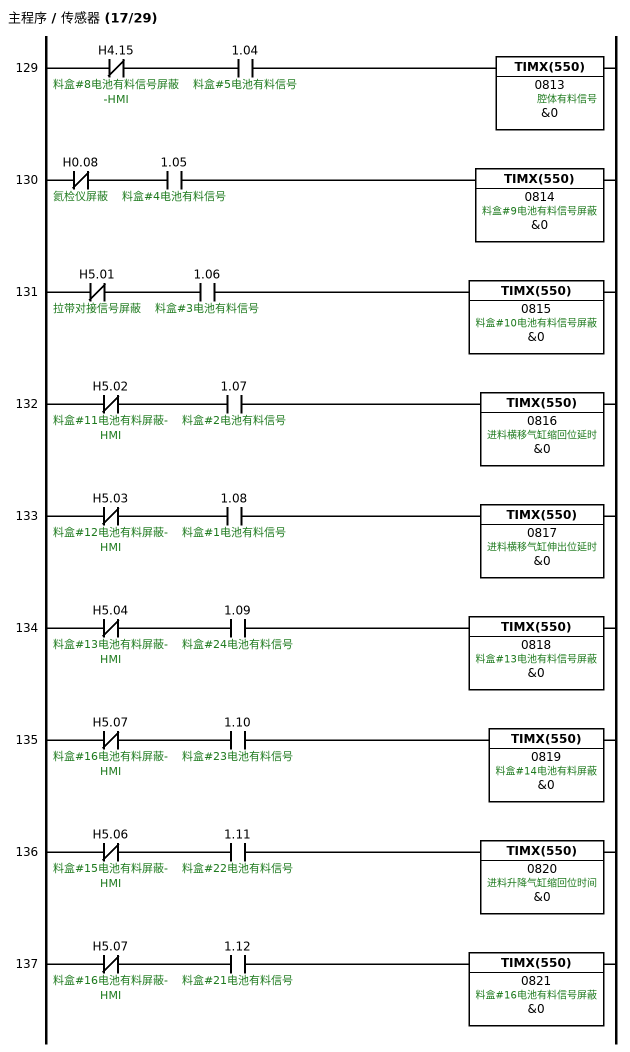
; [picture p24: 主程序 / 传感器, rungs 129-137]
; rung 129
LDNOT H4.15  ; 料盒#8电池有料信号屏蔽-HMI
AND 1.04  ; 料盒#5电池有料信号
TIMX(550) 0813 &0  ; 腔体有料信号
; rung 130
LDNOT H0.08  ; 氦检仪屏蔽
AND 1.05  ; 料盒#4电池有料信号
TIMX(550) 0814 &0  ; 料盒#9电池有料信号屏蔽
; rung 131
LDNOT H5.01  ; 拉带对接信号屏蔽
AND 1.06  ; 料盒#3电池有料信号
TIMX(550) 0815 &0  ; 料盒#10电池有料信号屏蔽
; rung 132
LDNOT H5.02  ; 料盒#11电池有料屏蔽-HMI
AND 1.07  ; 料盒#2电池有料信号
TIMX(550) 0816 &0  ; 进料横移气缸缩回位延时
; rung 133
LDNOT H5.03  ; 料盒#12电池有料屏蔽-HMI
AND 1.08  ; 料盒#1电池有料信号
TIMX(550) 0817 &0  ; 进料横移气缸伸出位延时
; rung 134
LDNOT H5.04  ; 料盒#13电池有料屏蔽-HMI
AND 1.09  ; 料盒#24电池有料信号
TIMX(550) 0818 &0  ; 料盒#13电池有料信号屏蔽
; rung 135
LDNOT H5.07  ; 料盒#16电池有料屏蔽-HMI
AND 1.10  ; 料盒#23电池有料信号
TIMX(550) 0819 &0  ; 料盒#14电池有料屏蔽
; rung 136
LDNOT H5.06  ; 料盒#15电池有料屏蔽-HMI
AND 1.11  ; 料盒#22电池有料信号
TIMX(550) 0820 &0  ; 进料升降气缸缩回位时间
; rung 137
LDNOT H5.07  ; 料盒#16电池有料屏蔽-HMI
AND 1.12  ; 料盒#21电池有料信号
TIMX(550) 0821 &0  ; 料盒#16电池有料信号屏蔽

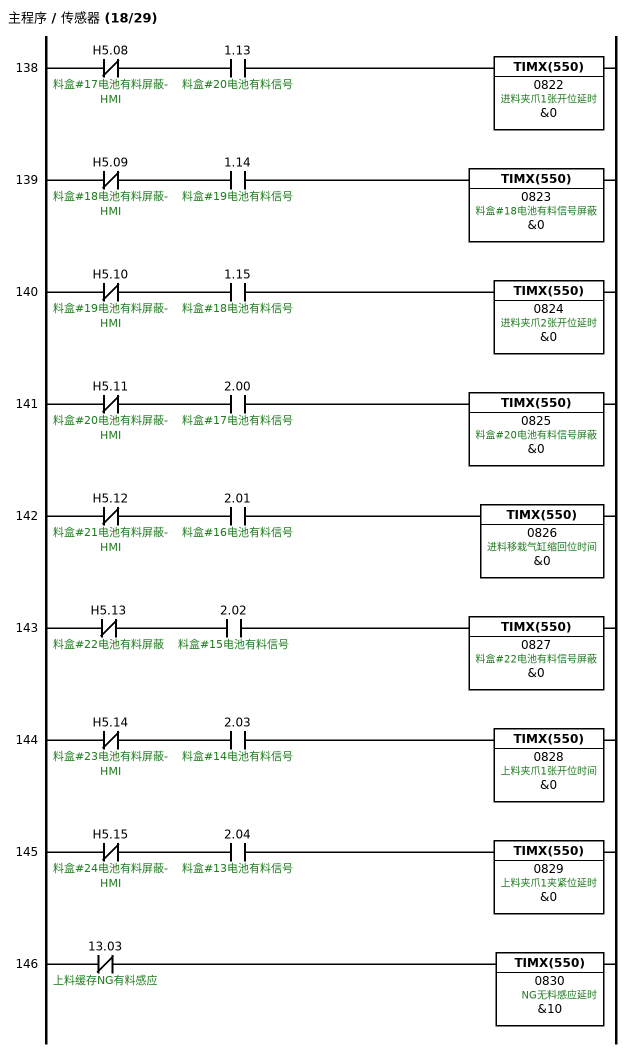
; rung 138
LDNOT H5.08  ; 料盒#17电池有料屏蔽-HMI
AND 1.13  ; 料盒#20电池有料信号
TIMX(550) 0822 &0  ; 进料夹爪1张开位延时
; rung 139
LDNOT H5.09  ; 料盒#18电池有料屏蔽-HMI
AND 1.14  ; 料盒#19电池有料信号
TIMX(550) 0823 &0  ; 料盒#18电池有料信号屏蔽
; rung 140
LDNOT H5.10  ; 料盒#19电池有料屏蔽-HMI
AND 1.15  ; 料盒#18电池有料信号
TIMX(550) 0824 &0  ; 进料夹爪2张开位延时
; rung 141
LDNOT H5.11  ; 料盒#20电池有料屏蔽-HMI
AND 2.00  ; 料盒#17电池有料信号
TIMX(550) 0825 &0  ; 料盒#20电池有料信号屏蔽
; rung 142
LDNOT H5.12  ; 料盒#21电池有料屏蔽-HMI
AND 2.01  ; 料盒#16电池有料信号
TIMX(550) 0826 &0  ; 进料移栽气缸缩回位时间
; rung 143
LDNOT H5.13  ; 料盒#22电池有料屏蔽
AND 2.02  ; 料盒#15电池有料信号
TIMX(550) 0827 &0  ; 料盒#22电池有料信号屏蔽
; rung 144
LDNOT H5.14  ; 料盒#23电池有料屏蔽-HMI
AND 2.03  ; 料盒#14电池有料信号
TIMX(550) 0828 &0  ; 上料夹爪1张开位时间
; rung 145
LDNOT H5.15  ; 料盒#24电池有料屏蔽-HMI
AND 2.04  ; 料盒#13电池有料信号
TIMX(550) 0829 &0  ; 上料夹爪1夹紧位延时
; rung 146
LDNOT 13.03  ; 上料缓存NG有料感应
TIMX(550) 0830 &10  ; NG无料感应延时

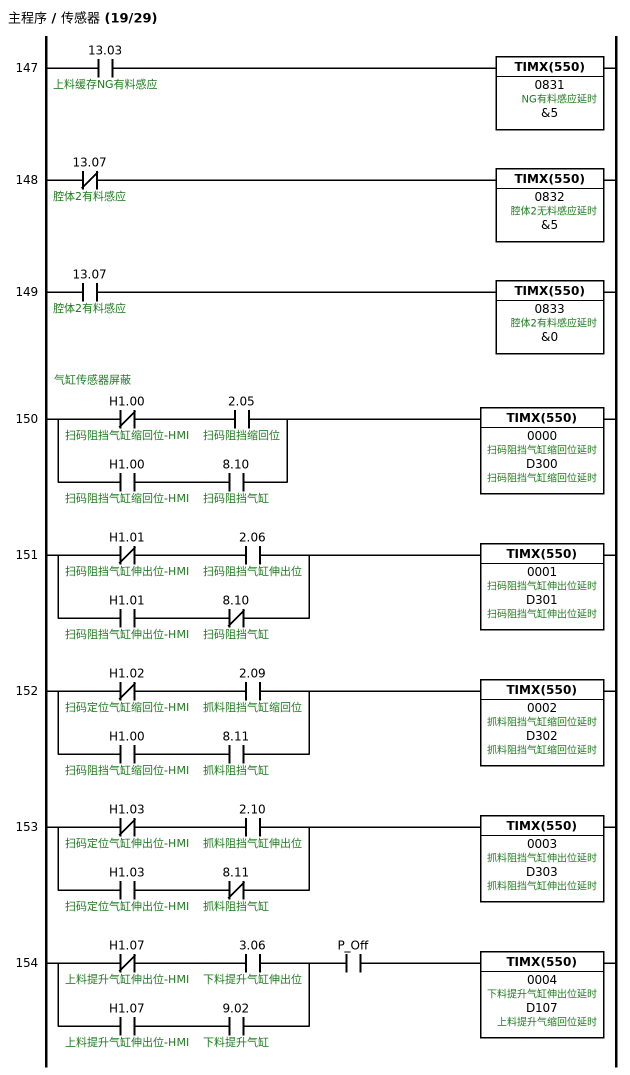
; rung 147
LD 13.03  ; 上料缓存NG有料感应
TIMX(550) 0831 &5  ; NG有料感应延时
; rung 148
LDNOT 13.07  ; 腔体2有料感应
TIMX(550) 0832 &5  ; 腔体2无料感应延时
; rung 149
LD 13.07  ; 腔体2有料感应
TIMX(550) 0833 &0  ; 腔体2有料感应延时
; rung 150: 气缸传感器屏蔽
LDNOT H1.00  ; 扫码阻挡气缸缩回位-HMI
AND 2.05  ; 扫码阻挡缩回位
LD H1.00  ; 扫码阻挡气缸缩回位-HMI
AND 8.10  ; 扫码阻挡气缸
ORLD
TIMX(550) 0000 D300  ; 扫码阻挡气缸缩回位延时
; rung 151
LDNOT H1.01  ; 扫码阻挡气缸伸出位-HMI
AND 2.06  ; 扫码阻挡气缸伸出位
LD H1.01  ; 扫码阻挡气缸伸出位-HMI
ANDNOT 8.10  ; 扫码阻挡气缸
ORLD
TIMX(550) 0001 D301  ; 扫码阻挡气缸伸出位延时
; rung 152
LDNOT H1.02  ; 扫码定位气缸缩回位-HMI
AND 2.09  ; 抓料阻挡气缸缩回位
LD H1.00  ; 扫码阻挡气缸缩回位-HMI
AND 8.11  ; 抓料阻挡气缸
ORLD
TIMX(550) 0002 D302  ; 抓料阻挡气缸缩回位延时
; rung 153
LDNOT H1.03  ; 扫码定位气缸伸出位-HMI
AND 2.10  ; 抓料阻挡气缸伸出位
LD H1.03  ; 扫码定位气缸伸出位-HMI
ANDNOT 8.11  ; 抓料阻挡气缸
ORLD
TIMX(550) 0003 D303  ; 抓料阻挡气缸伸出位延时
; rung 154
LDNOT H1.07  ; 上料提升气缸伸出位-HMI
AND 3.06  ; 下料提升气缸伸出位
LD H1.07  ; 上料提升气缸伸出位-HMI
AND 9.02  ; 下料提升气缸
ORLD
AND P_Off
TIMX(550) 0004 D107  ; 上料提升气缩回位延时, 下料提升气缸伸出位延时

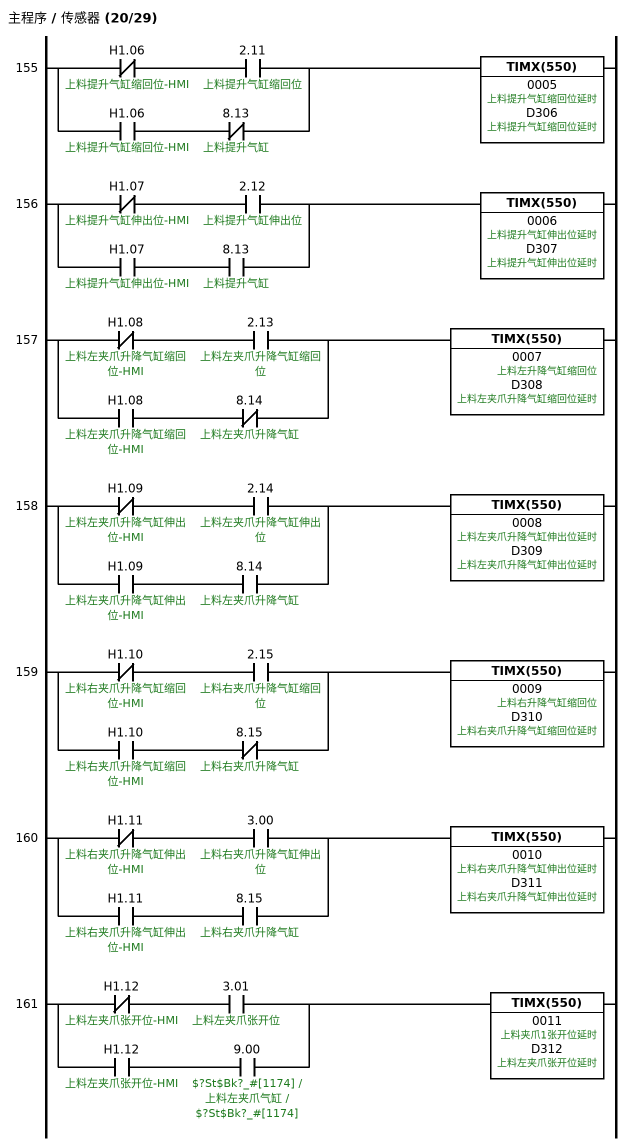
; rung 155
LDNOT H1.06  ; 上料提升气缸缩回位-HMI
AND 2.11  ; 上料提升气缸缩回位
LD H1.06  ; 上料提升气缸缩回位-HMI
ANDNOT 8.13  ; 上料提升气缸
ORLD
TIMX(550) 0005 D306  ; 上料提升气缸缩回位延时
; rung 156
LDNOT H1.07  ; 上料提升气缸伸出位-HMI
AND 2.12  ; 上料提升气缸伸出位
LD H1.07  ; 上料提升气缸伸出位-HMI
AND 8.13  ; 上料提升气缸
ORLD
TIMX(550) 0006 D307  ; 上料提升气缸伸出位延时
; rung 157
LDNOT H1.08  ; 上料左夹爪升降气缸缩回位-HMI
AND 2.13  ; 上料左夹爪升降气缸缩回位
LD H1.08  ; 上料左夹爪升降气缸缩回位-HMI
ANDNOT 8.14  ; 上料左夹爪升降气缸
ORLD
TIMX(550) 0007 D308  ; 上料左夹爪升降气缸缩回位延时, 上料左升降气缸缩回位
; rung 158
LDNOT H1.09  ; 上料左夹爪升降气缸伸出位-HMI
AND 2.14  ; 上料左夹爪升降气缸伸出位
LD H1.09  ; 上料左夹爪升降气缸伸出位-HMI
AND 8.14  ; 上料左夹爪升降气缸
ORLD
TIMX(550) 0008 D309  ; 上料左夹爪升降气缸伸出位延时
; rung 159
LDNOT H1.10  ; 上料右夹爪升降气缸缩回位-HMI
AND 2.15  ; 上料右夹爪升降气缸缩回位
LD H1.10  ; 上料右夹爪升降气缸缩回位-HMI
ANDNOT 8.15  ; 上料右夹爪升降气缸
ORLD
TIMX(550) 0009 D310  ; 上料右夹爪升降气缸缩回位延时, 上料右升降气缸缩回位
; rung 160
LDNOT H1.11  ; 上料右夹爪升降气缸伸出位-HMI
AND 3.00  ; 上料右夹爪升降气缸伸出位
LD H1.11  ; 上料右夹爪升降气缸伸出位-HMI
AND 8.15  ; 上料右夹爪升降气缸
ORLD
TIMX(550) 0010 D311  ; 上料右夹爪升降气缸伸出位延时
; rung 161
LDNOT H1.12  ; 上料左夹爪张开位-HMI
AND 3.01  ; 上料左夹爪张开位
LD H1.12  ; 上料左夹爪张开位-HMI
AND 9.00  ; $?St$Bk?_#[1174] / 上料左夹爪气缸 / $?St$Bk?_#[1174]
ORLD
TIMX(550) 0011 D312  ; 上料左夹爪张开位延时, 上料夹爪1张开位延时

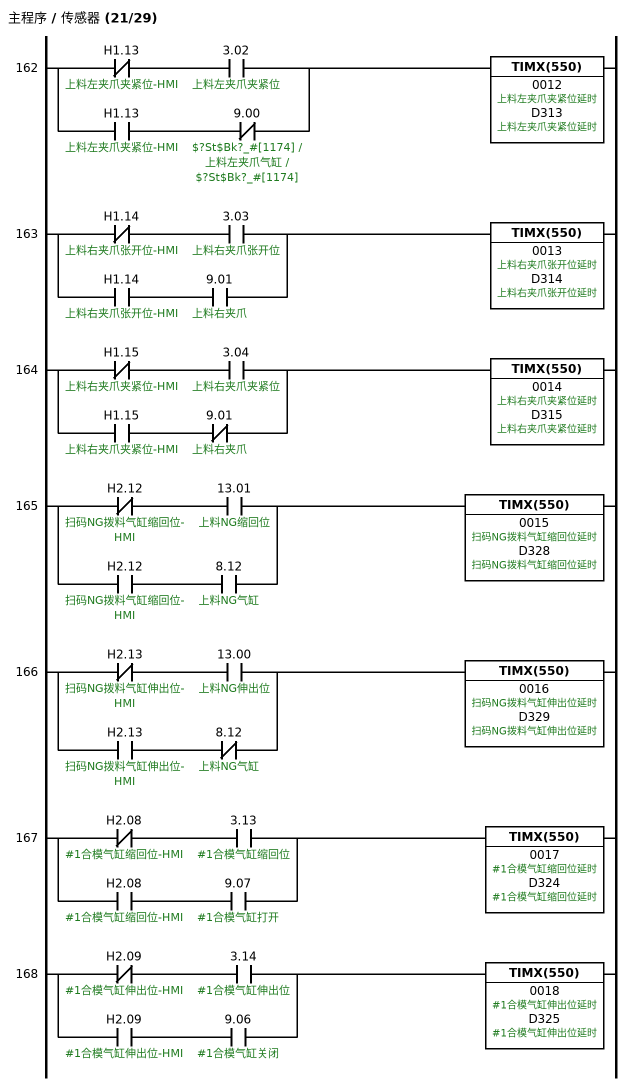
; rung 162
LDNOT H1.13  ; 上料左夹爪夹紧位-HMI
AND 3.02  ; 上料左夹爪夹紧位
LD H1.13  ; 上料左夹爪夹紧位-HMI
ANDNOT 9.00  ; $?St$Bk?_#[1174] / 上料左夹爪气缸 / $?St$Bk?_#[1174]
ORLD
TIMX(550) 0012 D313  ; 上料左夹爪夹紧位延时
; rung 163
LDNOT H1.14  ; 上料右夹爪张开位-HMI
AND 3.03  ; 上料右夹爪张开位
LD H1.14  ; 上料右夹爪张开位-HMI
AND 9.01  ; 上料右夹爪
ORLD
TIMX(550) 0013 D314  ; 上料右夹爪张开位延时
; rung 164
LDNOT H1.15  ; 上料右夹爪夹紧位-HMI
AND 3.04  ; 上料右夹爪夹紧位
LD H1.15  ; 上料右夹爪夹紧位-HMI
ANDNOT 9.01  ; 上料右夹爪
ORLD
TIMX(550) 0014 D315  ; 上料右夹爪夹紧位延时
; rung 165
LDNOT H2.12  ; 扫码NG拨料气缸缩回位-HMI
AND 13.01  ; 上料NG缩回位
LD H2.12  ; 扫码NG拨料气缸缩回位-HMI
AND 8.12  ; 上料NG气缸
ORLD
TIMX(550) 0015 D328  ; 扫码NG拨料气缸缩回位延时
; rung 166
LDNOT H2.13  ; 扫码NG拨料气缸伸出位-HMI
AND 13.00  ; 上料NG伸出位
LD H2.13  ; 扫码NG拨料气缸伸出位-HMI
ANDNOT 8.12  ; 上料NG气缸
ORLD
TIMX(550) 0016 D329  ; 扫码NG拨料气缸伸出位延时
; rung 167
LDNOT H2.08  ; #1合模气缸缩回位-HMI
AND 3.13  ; #1合模气缸缩回位
LD H2.08  ; #1合模气缸缩回位-HMI
AND 9.07  ; #1合模气缸打开
ORLD
TIMX(550) 0017 D324  ; #1合模气缸缩回位延时
; rung 168
LDNOT H2.09  ; #1合模气缸伸出位-HMI
AND 3.14  ; #1合模气缸伸出位
LD H2.09  ; #1合模气缸伸出位-HMI
AND 9.06  ; #1合模气缸关闭
ORLD
TIMX(550) 0018 D325  ; #1合模气缸伸出位延时

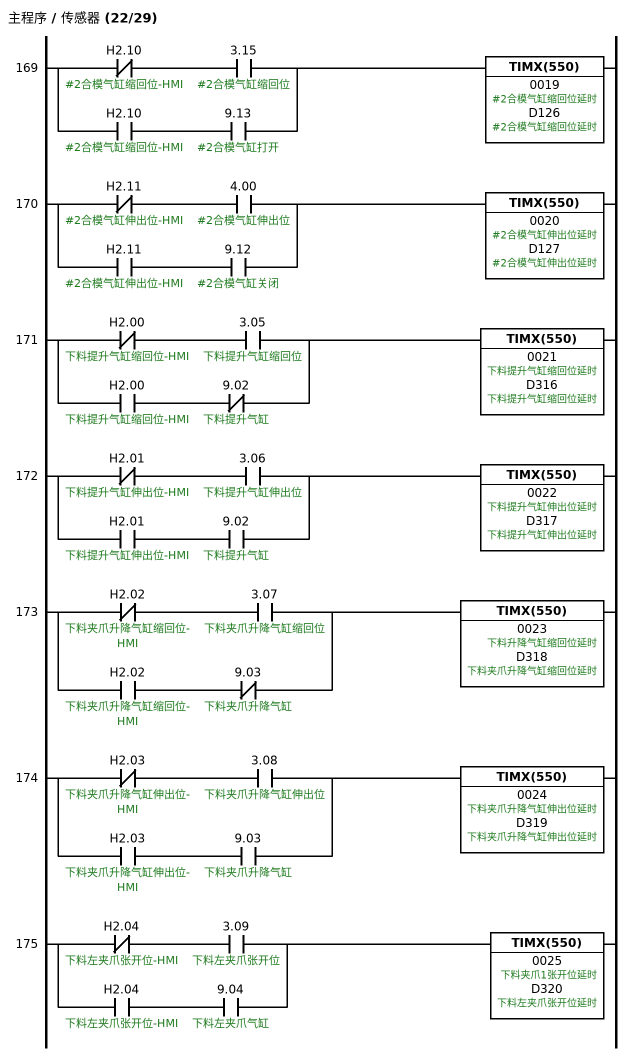
; rung 169
LDNOT H2.10  ; #2合模气缸缩回位-HMI
AND 3.15  ; #2合模气缸缩回位
LD H2.10  ; #2合模气缸缩回位-HMI
AND 9.13  ; #2合模气缸打开
ORLD
TIMX(550) 0019 D126  ; #2合模气缸缩回位延时
; rung 170
LDNOT H2.11  ; #2合模气缸伸出位-HMI
AND 4.00  ; #2合模气缸伸出位
LD H2.11  ; #2合模气缸伸出位-HMI
AND 9.12  ; #2合模气缸关闭
ORLD
TIMX(550) 0020 D127  ; #2合模气缸伸出位延时
; rung 171
LDNOT H2.00  ; 下料提升气缸缩回位-HMI
AND 3.05  ; 下料提升气缸缩回位
LD H2.00  ; 下料提升气缸缩回位-HMI
ANDNOT 9.02  ; 下料提升气缸
ORLD
TIMX(550) 0021 D316  ; 下料提升气缸缩回位延时
; rung 172
LDNOT H2.01  ; 下料提升气缸伸出位-HMI
AND 3.06  ; 下料提升气缸伸出位
LD H2.01  ; 下料提升气缸伸出位-HMI
AND 9.02  ; 下料提升气缸
ORLD
TIMX(550) 0022 D317  ; 下料提升气缸伸出位延时
; rung 173
LDNOT H2.02  ; 下料夹爪升降气缸缩回位-HMI
AND 3.07  ; 下料夹爪升降气缸缩回位
LD H2.02  ; 下料夹爪升降气缸缩回位-HMI
ANDNOT 9.03  ; 下料夹爪升降气缸
ORLD
TIMX(550) 0023 D318  ; 下料夹爪升降气缸缩回位延时, 下料升降气缸缩回位延时
; rung 174
LDNOT H2.03  ; 下料夹爪升降气缸伸出位-HMI
AND 3.08  ; 下料夹爪升降气缸伸出位
LD H2.03  ; 下料夹爪升降气缸伸出位-HMI
AND 9.03  ; 下料夹爪升降气缸
ORLD
TIMX(550) 0024 D319  ; 下料夹爪升降气缸伸出位延时
; rung 175
LDNOT H2.04  ; 下料左夹爪张开位-HMI
AND 3.09  ; 下料左夹爪张开位
LD H2.04  ; 下料左夹爪张开位-HMI
AND 9.04  ; 下料左夹爪气缸
ORLD
TIMX(550) 0025 D320  ; 下料左夹爪张开位延时, 下料夹爪1张开位延时

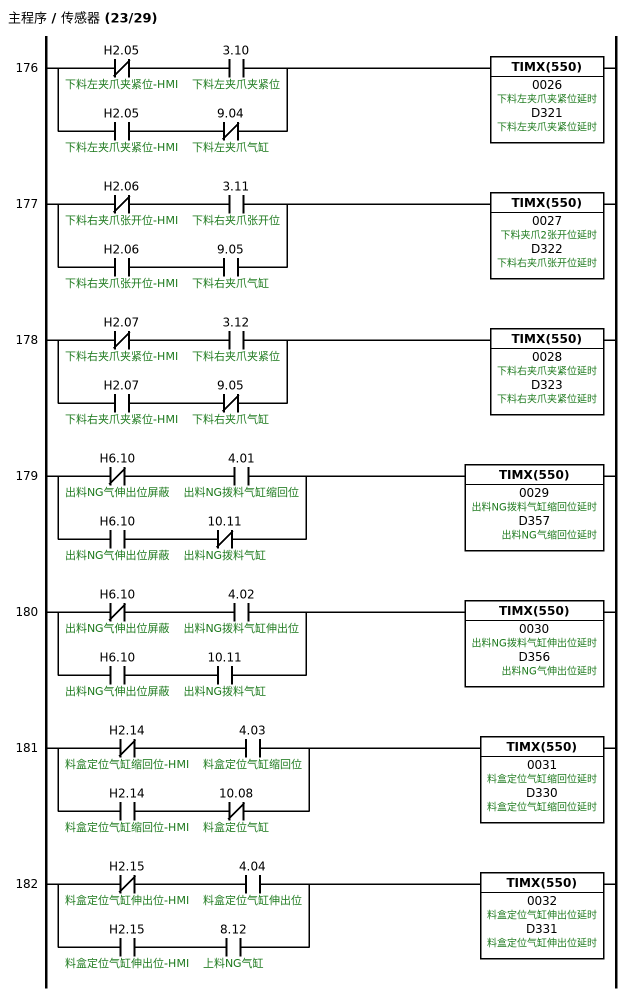
; rung 176
LDNOT H2.05  ; 下料左夹爪夹紧位-HMI
AND 3.10  ; 下料左夹爪夹紧位
LD H2.05  ; 下料左夹爪夹紧位-HMI
ANDNOT 9.04  ; 下料左夹爪气缸
ORLD
TIMX(550) 0026 D321  ; 下料左夹爪夹紧位延时
; rung 177
LDNOT H2.06  ; 下料右夹爪张开位-HMI
AND 3.11  ; 下料右夹爪张开位
LD H2.06  ; 下料右夹爪张开位-HMI
AND 9.05  ; 下料右夹爪气缸
ORLD
TIMX(550) 0027 D322  ; 下料右夹爪张开位延时, 下料夹爪2张开位延时
; rung 178
LDNOT H2.07  ; 下料右夹爪夹紧位-HMI
AND 3.12  ; 下料右夹爪夹紧位
LD H2.07  ; 下料右夹爪夹紧位-HMI
ANDNOT 9.05  ; 下料右夹爪气缸
ORLD
TIMX(550) 0028 D323  ; 下料右夹爪夹紧位延时
; rung 179
LDNOT H6.10  ; 出料NG气伸出位屏蔽
AND 4.01  ; 出料NG拨料气缸缩回位
LD H6.10  ; 出料NG气伸出位屏蔽
ANDNOT 10.11  ; 出料NG拨料气缸
ORLD
TIMX(550) 0029 D357  ; 出料NG气缩回位延时, 出料NG拨料气缸缩回位延时
; rung 180
LDNOT H6.10  ; 出料NG气伸出位屏蔽
AND 4.02  ; 出料NG拨料气缸伸出位
LD H6.10  ; 出料NG气伸出位屏蔽
AND 10.11  ; 出料NG拨料气缸
ORLD
TIMX(550) 0030 D356  ; 出料NG气伸出位延时, 出料NG拨料气缸伸出位延时
; rung 181
LDNOT H2.14  ; 料盒定位气缸缩回位-HMI
AND 4.03  ; 料盒定位气缸缩回位
LD H2.14  ; 料盒定位气缸缩回位-HMI
ANDNOT 10.08  ; 料盒定位气缸
ORLD
TIMX(550) 0031 D330  ; 料盒定位气缸缩回位延时
; rung 182
LDNOT H2.15  ; 料盒定位气缸伸出位-HMI
AND 4.04  ; 料盒定位气缸伸出位
LD H2.15  ; 料盒定位气缸伸出位-HMI
AND 8.12  ; 上料NG气缸
ORLD
TIMX(550) 0032 D331  ; 料盒定位气缸伸出位延时

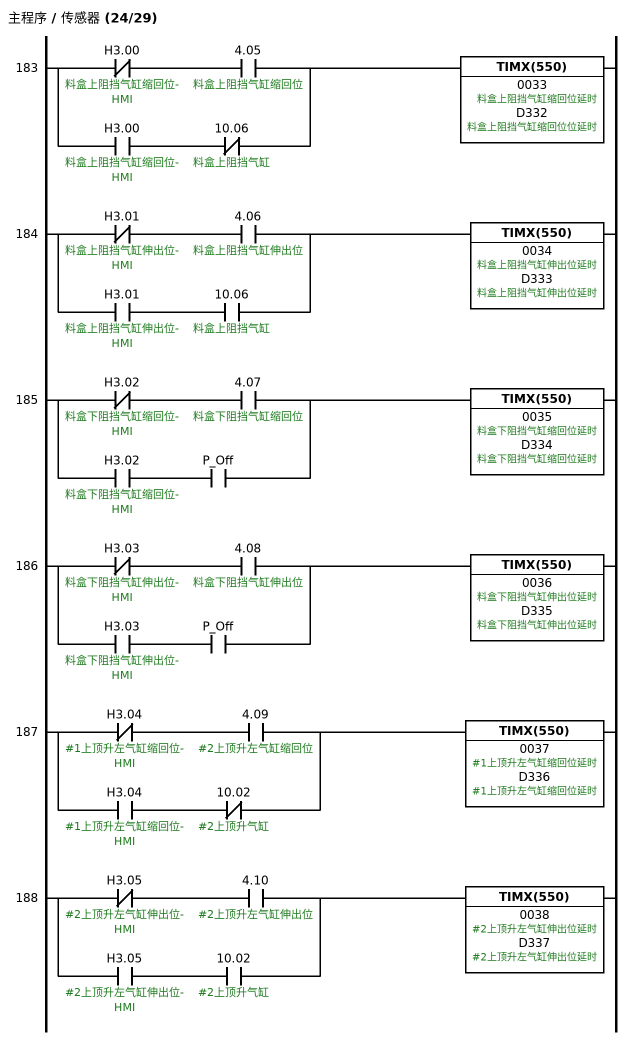
; rung 183
LDNOT H3.00  ; 料盒上阻挡气缸缩回位-HMI
AND 4.05  ; 料盒上阻挡气缸缩回位
LD H3.00  ; 料盒上阻挡气缸缩回位-HMI
ANDNOT 10.06  ; 料盒上阻挡气缸
ORLD
TIMX(550) 0033 D332  ; 料盒上阻挡气缸缩回位位延时, 料盒上阻挡气缸缩回位延时
; rung 184
LDNOT H3.01  ; 料盒上阻挡气缸伸出位-HMI
AND 4.06  ; 料盒上阻挡气缸伸出位
LD H3.01  ; 料盒上阻挡气缸伸出位-HMI
AND 10.06  ; 料盒上阻挡气缸
ORLD
TIMX(550) 0034 D333  ; 料盒上阻挡气缸伸出位延时
; rung 185
LDNOT H3.02  ; 料盒下阻挡气缸缩回位-HMI
AND 4.07  ; 料盒下阻挡气缸缩回位
LD H3.02  ; 料盒下阻挡气缸缩回位-HMI
AND P_Off
ORLD
TIMX(550) 0035 D334  ; 料盒下阻挡气缸缩回位延时
; rung 186
LDNOT H3.03  ; 料盒下阻挡气缸伸出位-HMI
AND 4.08  ; 料盒下阻挡气缸伸出位
LD H3.03  ; 料盒下阻挡气缸伸出位-HMI
AND P_Off
ORLD
TIMX(550) 0036 D335  ; 料盒下阻挡气缸伸出位延时
; rung 187
LDNOT H3.04  ; #1上顶升左气缸缩回位-HMI
AND 4.09  ; #2上顶升左气缸缩回位
LD H3.04  ; #1上顶升左气缸缩回位-HMI
ANDNOT 10.02  ; #2上顶升气缸
ORLD
TIMX(550) 0037 D336  ; #1上顶升左气缸缩回位延时
; rung 188
LDNOT H3.05  ; #2上顶升左气缸伸出位-HMI
AND 4.10  ; #2上顶升左气缸伸出位
LD H3.05  ; #2上顶升左气缸伸出位-HMI
AND 10.02  ; #2上顶升气缸
ORLD
TIMX(550) 0038 D337  ; #2上顶升左气缸伸出位延时

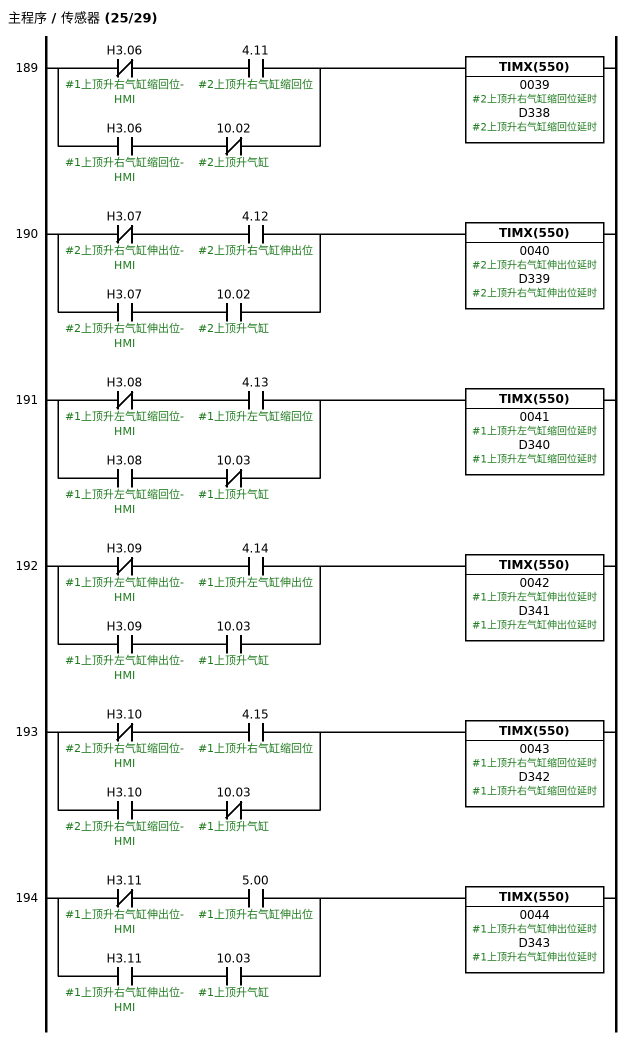
; rung 189
LDNOT H3.06  ; #1上顶升右气缸缩回位-HMI
AND 4.11  ; #2上顶升右气缸缩回位
LD H3.06  ; #1上顶升右气缸缩回位-HMI
ANDNOT 10.02  ; #2上顶升气缸
ORLD
TIMX(550) 0039 D338  ; #2上顶升右气缸缩回位延时
; rung 190
LDNOT H3.07  ; #2上顶升右气缸伸出位-HMI
AND 4.12  ; #2上顶升右气缸伸出位
LD H3.07  ; #2上顶升右气缸伸出位-HMI
AND 10.02  ; #2上顶升气缸
ORLD
TIMX(550) 0040 D339  ; #2上顶升右气缸伸出位延时
; rung 191
LDNOT H3.08  ; #1上顶升左气缸缩回位-HMI
AND 4.13  ; #1上顶升左气缸缩回位
LD H3.08  ; #1上顶升左气缸缩回位-HMI
ANDNOT 10.03  ; #1上顶升气缸
ORLD
TIMX(550) 0041 D340  ; #1上顶升左气缸缩回位延时
; rung 192
LDNOT H3.09  ; #1上顶升左气缸伸出位-HMI
AND 4.14  ; #1上顶升左气缸伸出位
LD H3.09  ; #1上顶升左气缸伸出位-HMI
AND 10.03  ; #1上顶升气缸
ORLD
TIMX(550) 0042 D341  ; #1上顶升左气缸伸出位延时
; rung 193
LDNOT H3.10  ; #2上顶升右气缸缩回位-HMI
AND 4.15  ; #1上顶升右气缸缩回位
LD H3.10  ; #2上顶升右气缸缩回位-HMI
ANDNOT 10.03  ; #1上顶升气缸
ORLD
TIMX(550) 0043 D342  ; #1上顶升右气缸缩回位延时
; rung 194
LDNOT H3.11  ; #1上顶升右气缸伸出位-HMI
AND 5.00  ; #1上顶升右气缸伸出位
LD H3.11  ; #1上顶升右气缸伸出位-HMI
AND 10.03  ; #1上顶升气缸
ORLD
TIMX(550) 0044 D343  ; #1上顶升右气缸伸出位延时

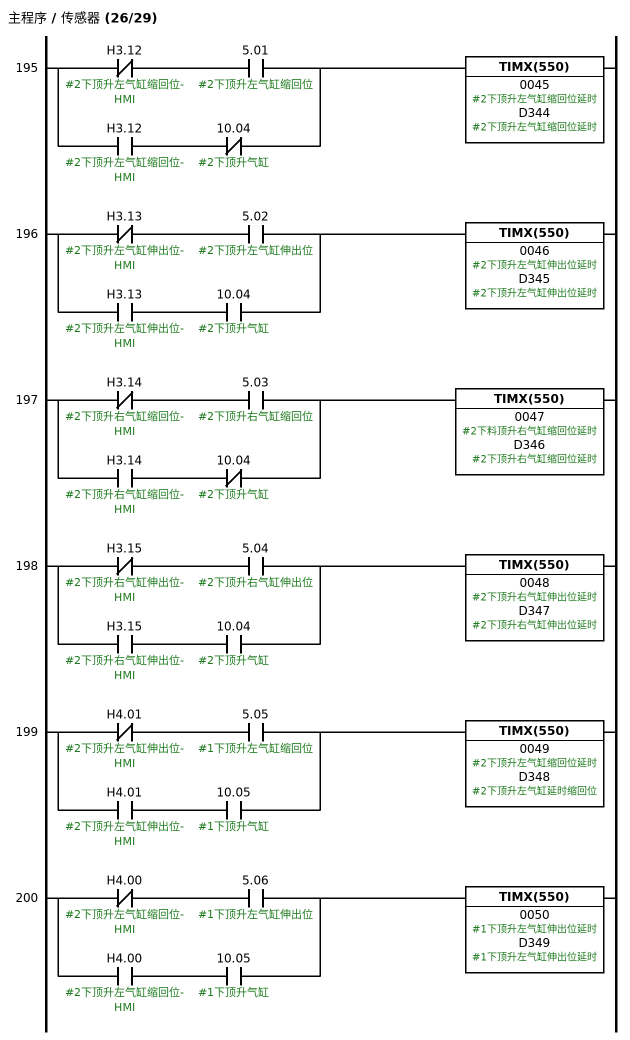
; rung 195
LDNOT H3.12  ; #2下顶升左气缸缩回位-HMI
AND 5.01  ; #2下顶升左气缸缩回位
LD H3.12  ; #2下顶升左气缸缩回位-HMI
ANDNOT 10.04  ; #2下顶升气缸
ORLD
TIMX(550) 0045 D344  ; #2下顶升左气缸缩回位延时
; rung 196
LDNOT H3.13  ; #2下顶升左气缸伸出位-HMI
AND 5.02  ; #2下顶升左气缸伸出位
LD H3.13  ; #2下顶升左气缸伸出位-HMI
AND 10.04  ; #2下顶升气缸
ORLD
TIMX(550) 0046 D345  ; #2下顶升左气缸伸出位延时
; rung 197
LDNOT H3.14  ; #2下顶升右气缸缩回位-HMI
AND 5.03  ; #2下顶升右气缸缩回位
LD H3.14  ; #2下顶升右气缸缩回位-HMI
ANDNOT 10.04  ; #2下顶升气缸
ORLD
TIMX(550) 0047 D346  ; #2下顶升右气缸缩回位延时, #2下料顶升右气缸缩回位延时
; rung 198
LDNOT H3.15  ; #2下顶升右气缸伸出位-HMI
AND 5.04  ; #2下顶升右气缸伸出位
LD H3.15  ; #2下顶升右气缸伸出位-HMI
AND 10.04  ; #2下顶升气缸
ORLD
TIMX(550) 0048 D347  ; #2下顶升右气缸伸出位延时
; rung 199
LDNOT H4.01  ; #2下顶升左气缸伸出位-HMI
AND 5.05  ; #1下顶升左气缸缩回位
LD H4.01  ; #2下顶升左气缸伸出位-HMI
AND 10.05  ; #1下顶升气缸
ORLD
TIMX(550) 0049 D348  ; #2下顶升左气缸延时缩回位, #2下顶升左气缸缩回位延时
; rung 200
LDNOT H4.00  ; #2下顶升左气缸缩回位-HMI
AND 5.06  ; #1下顶升左气缸伸出位
LD H4.00  ; #2下顶升左气缸缩回位-HMI
AND 10.05  ; #1下顶升气缸
ORLD
TIMX(550) 0050 D349  ; #1下顶升左气缸伸出位延时

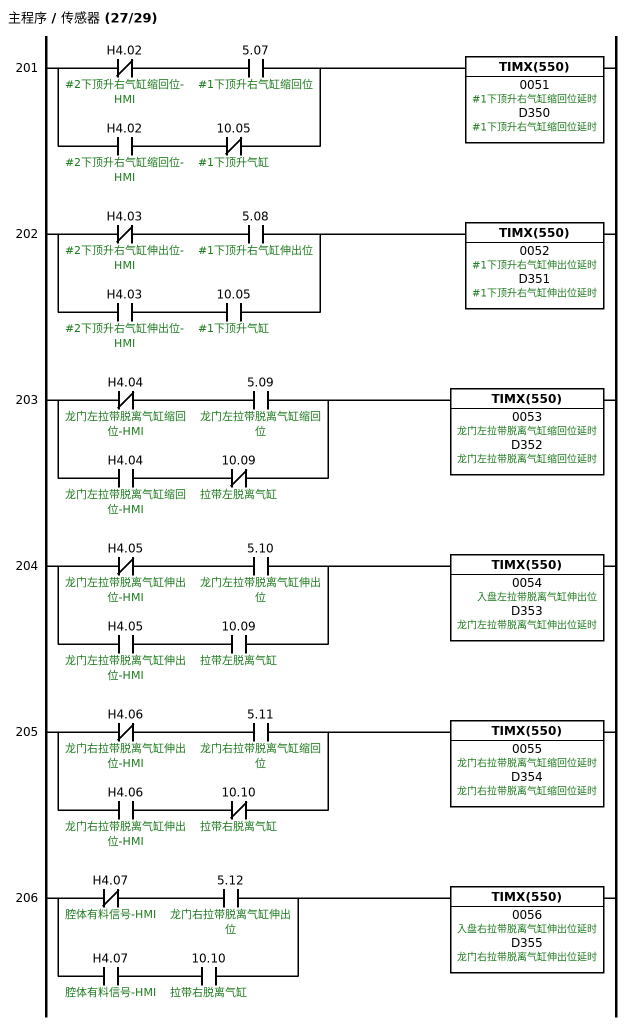
; rung 201
LDNOT H4.02  ; #2下顶升右气缸缩回位-HMI
AND 5.07  ; #1下顶升右气缸缩回位
LD H4.02  ; #2下顶升右气缸缩回位-HMI
ANDNOT 10.05  ; #1下顶升气缸
ORLD
TIMX(550) 0051 D350  ; #1下顶升右气缸缩回位延时
; rung 202
LDNOT H4.03  ; #2下顶升右气缸伸出位-HMI
AND 5.08  ; #1下顶升右气缸伸出位
LD H4.03  ; #2下顶升右气缸伸出位-HMI
AND 10.05  ; #1下顶升气缸
ORLD
TIMX(550) 0052 D351  ; #1下顶升右气缸伸出位延时
; rung 203
LDNOT H4.04  ; 龙门左拉带脱离气缸缩回位-HMI
AND 5.09  ; 龙门左拉带脱离气缸缩回位
LD H4.04  ; 龙门左拉带脱离气缸缩回位-HMI
ANDNOT 10.09  ; 拉带左脱离气缸
ORLD
TIMX(550) 0053 D352  ; 龙门左拉带脱离气缸缩回位延时
; rung 204
LDNOT H4.05  ; 龙门左拉带脱离气缸伸出位-HMI
AND 5.10  ; 龙门左拉带脱离气缸伸出位
LD H4.05  ; 龙门左拉带脱离气缸伸出位-HMI
AND 10.09  ; 拉带左脱离气缸
ORLD
TIMX(550) 0054 D353  ; 龙门左拉带脱离气缸伸出位延时, 入盘左拉带脱离气缸伸出位
; rung 205
LDNOT H4.06  ; 龙门右拉带脱离气缸伸出位-HMI
AND 5.11  ; 龙门右拉带脱离气缸缩回位
LD H4.06  ; 龙门右拉带脱离气缸伸出位-HMI
ANDNOT 10.10  ; 拉带右脱离气缸
ORLD
TIMX(550) 0055 D354  ; 龙门右拉带脱离气缸缩回位延时
; rung 206
LDNOT H4.07  ; 腔体有料信号-HMI
AND 5.12  ; 龙门右拉带脱离气缸伸出位
LD H4.07  ; 腔体有料信号-HMI
AND 10.10  ; 拉带右脱离气缸
ORLD
TIMX(550) 0056 D355  ; 龙门右拉带脱离气缸伸出位延时, 入盘右拉带脱离气缸伸出位延时

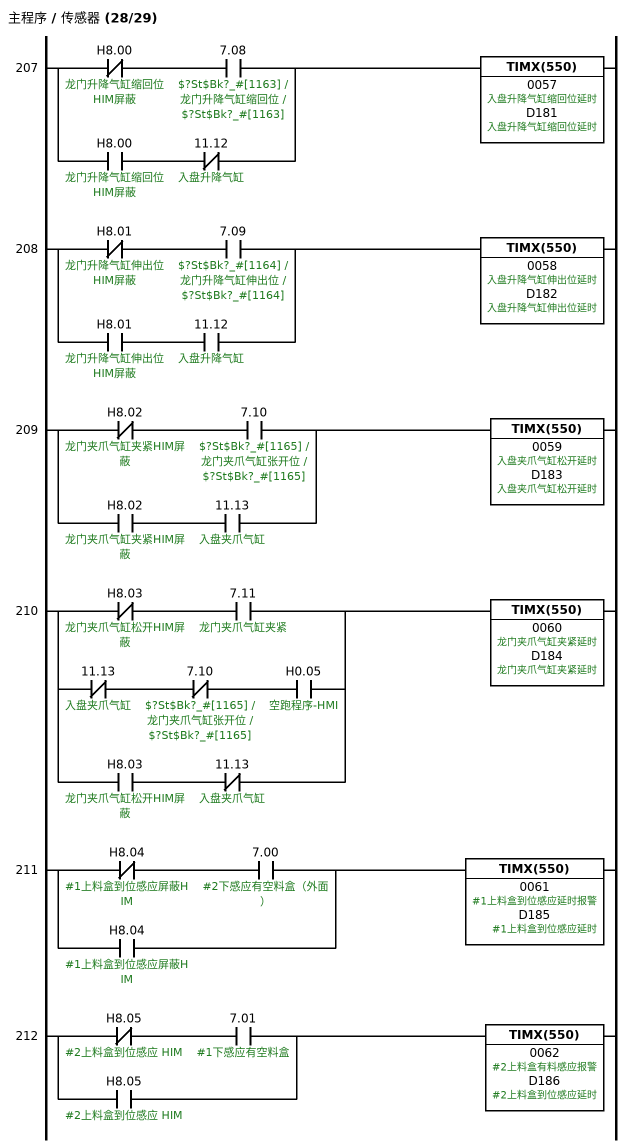
; rung 207
LDNOT H8.00  ; 龙门升降气缸缩回位 HIM屏蔽
AND 7.08  ; $?St$Bk?_#[1163] / 龙门升降气缸缩回位 / $?St$Bk?_#[1163]
LD H8.00  ; 龙门升降气缸缩回位 HIM屏蔽
ANDNOT 11.12  ; 入盘升降气缸
ORLD
TIMX(550) 0057 D181  ; 入盘升降气缸缩回位延时
; rung 208
LDNOT H8.01  ; 龙门升降气缸伸出位 HIM屏蔽
AND 7.09  ; $?St$Bk?_#[1164] / 龙门升降气缸伸出位 / $?St$Bk?_#[1164]
LD H8.01  ; 龙门升降气缸伸出位 HIM屏蔽
AND 11.12  ; 入盘升降气缸
ORLD
TIMX(550) 0058 D182  ; 入盘升降气缸伸出位延时
; rung 209
LDNOT H8.02  ; 龙门夹爪气缸夹紧HIM屏蔽
AND 7.10  ; $?St$Bk?_#[1165] / 龙门夹爪气缸张开位 / $?St$Bk?_#[1165]
LD H8.02  ; 龙门夹爪气缸夹紧HIM屏蔽
AND 11.13  ; 入盘夹爪气缸
ORLD
TIMX(550) 0059 D183  ; 入盘夹爪气缸松开延时
; rung 210
LDNOT H8.03  ; 龙门夹爪气缸松开HIM屏蔽
AND 7.11  ; 龙门夹爪气缸夹紧
LDNOT 11.13  ; 入盘夹爪气缸
ANDNOT 7.10  ; $?St$Bk?_#[1165] / 龙门夹爪气缸张开位 / $?St$Bk?_#[1165]
AND H0.05  ; 空跑程序-HMI
ORLD
LD H8.03  ; 龙门夹爪气缸松开HIM屏蔽
ANDNOT 11.13  ; 入盘夹爪气缸
ORLD
TIMX(550) 0060 D184  ; 龙门夹爪气缸夹紧延时
; rung 211
LDNOT H8.04  ; #1上料盒到位感应屏蔽HIM
AND 7.00  ; #2下感应有空料盒（外面）
OR H8.04  ; #1上料盒到位感应屏蔽HIM
TIMX(550) 0061 D185  ; #1上料盒到位感应延时, #1上料盒到位感应延时报警
; rung 212
LDNOT H8.05  ; #2上料盒到位感应 HIM
AND 7.01  ; #1下感应有空料盒
OR H8.05  ; #2上料盒到位感应 HIM
TIMX(550) 0062 D186  ; #2上料盒到位感应延时, #2上料盒有料感应报警

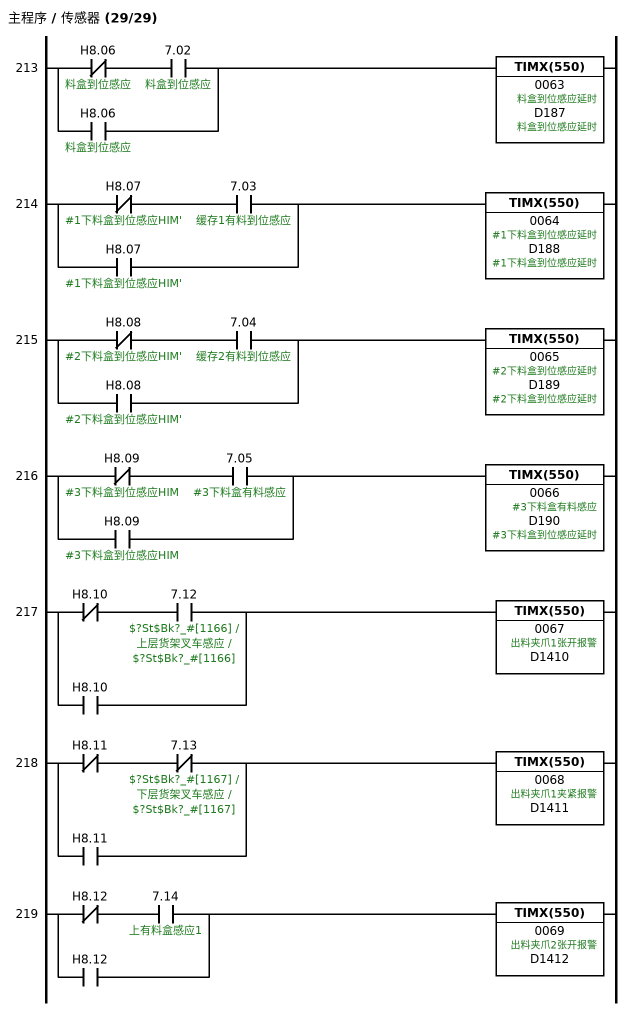
; rung 213
LDNOT H8.06  ; 料盒到位感应
AND 7.02  ; 料盒到位感应
OR H8.06  ; 料盒到位感应
TIMX(550) 0063 D187  ; 料盒到位感应延时
; rung 214
LDNOT H8.07  ; #1下料盒到位感应HIM'
AND 7.03  ; 缓存1有料到位感应
OR H8.07  ; #1下料盒到位感应HIM'
TIMX(550) 0064 D188  ; #1下料盒到位感应延时
; rung 215
LDNOT H8.08  ; #2下料盒到位感应HIM'
AND 7.04  ; 缓存2有料到位感应
OR H8.08  ; #2下料盒到位感应HIM'
TIMX(550) 0065 D189  ; #2下料盒到位感应延时
; rung 216
LDNOT H8.09  ; #3下料盒到位感应HIM
AND 7.05  ; #3下料盒有料感应
OR H8.09  ; #3下料盒到位感应HIM
TIMX(550) 0066 D190  ; #3下料盒到位感应延时, #3下料盒有料感应
; rung 217
LDNOT H8.10
AND 7.12  ; $?St$Bk?_#[1166] / 上层货架叉车感应 / $?St$Bk?_#[1166]
OR H8.10
TIMX(550) 0067 D1410  ; 出料夹爪1张开报警
; rung 218
LDNOT H8.11
ANDNOT 7.13  ; $?St$Bk?_#[1167] / 下层货架叉车感应 / $?St$Bk?_#[1167]
OR H8.11
TIMX(550) 0068 D1411  ; 出料夹爪1夹紧报警
; rung 219
LDNOT H8.12
AND 7.14  ; 上有料盒感应1
OR H8.12
TIMX(550) 0069 D1412  ; 出料夹爪2张开报警

### Section 超时判断

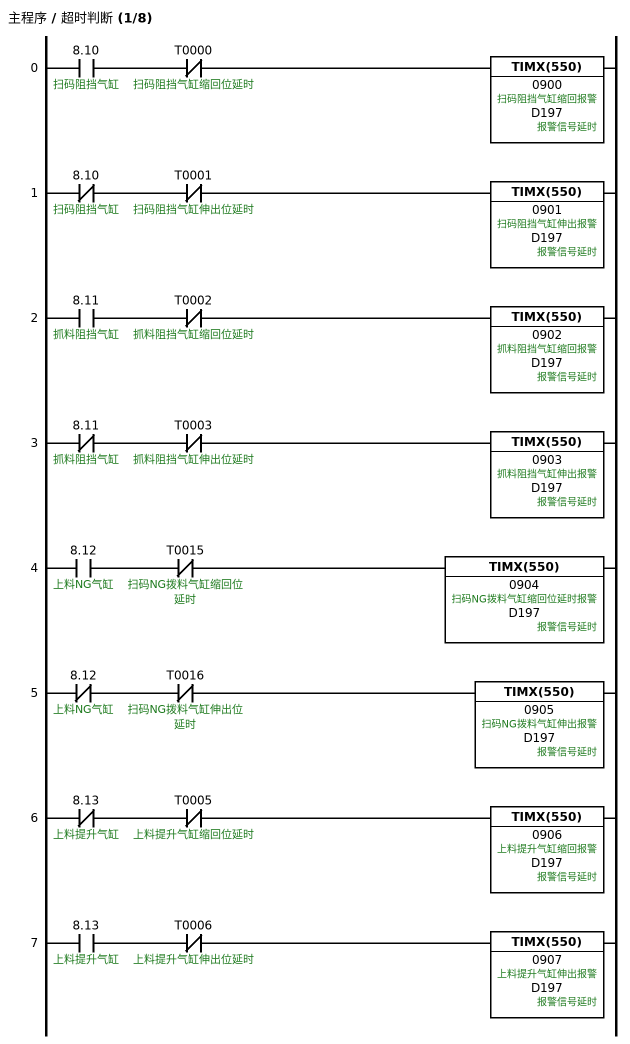
; rung 0
LD 8.10  ; 扫码阻挡气缸
ANDNOT T0000  ; 扫码阻挡气缸缩回位延时
TIMX(550) 0900 D197  ; 报警信号延时, 扫码阻挡气缸缩回报警
; rung 1
LDNOT 8.10  ; 扫码阻挡气缸
ANDNOT T0001  ; 扫码阻挡气缸伸出位延时
TIMX(550) 0901 D197  ; 报警信号延时, 扫码阻挡气缸伸出报警
; rung 2
LD 8.11  ; 抓料阻挡气缸
ANDNOT T0002  ; 抓料阻挡气缸缩回位延时
TIMX(550) 0902 D197  ; 报警信号延时, 抓料阻挡气缸缩回报警
; rung 3
LDNOT 8.11  ; 抓料阻挡气缸
ANDNOT T0003  ; 抓料阻挡气缸伸出位延时
TIMX(550) 0903 D197  ; 报警信号延时, 抓料阻挡气缸伸出报警
; rung 4
LD 8.12  ; 上料NG气缸
ANDNOT T0015  ; 扫码NG拨料气缸缩回位延时
TIMX(550) 0904 D197  ; 报警信号延时, 扫码NG拨料气缸缩回位延时报警
; rung 5
LDNOT 8.12  ; 上料NG气缸
ANDNOT T0016  ; 扫码NG拨料气缸伸出位延时
TIMX(550) 0905 D197  ; 报警信号延时, 扫码NG拨料气缸伸出报警
; rung 6
LDNOT 8.13  ; 上料提升气缸
ANDNOT T0005  ; 上料提升气缸缩回位延时
TIMX(550) 0906 D197  ; 报警信号延时, 上料提升气缸缩回报警
; rung 7
LD 8.13  ; 上料提升气缸
ANDNOT T0006  ; 上料提升气缸伸出位延时
TIMX(550) 0907 D197  ; 报警信号延时, 上料提升气缸伸出报警

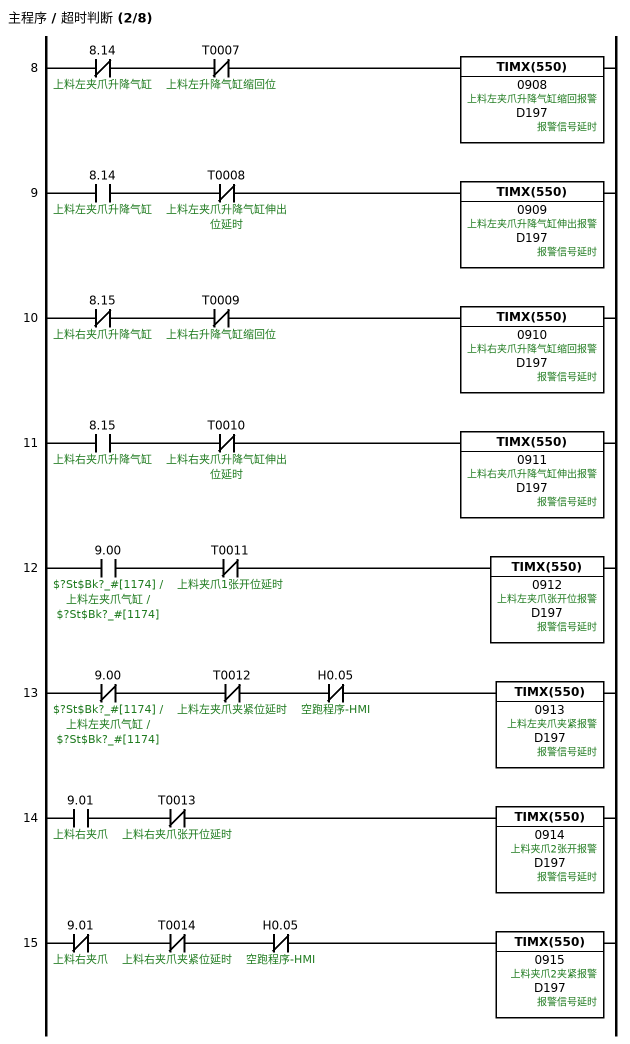
; rung 8
LDNOT 8.14  ; 上料左夹爪升降气缸
ANDNOT T0007  ; 上料左升降气缸缩回位
TIMX(550) 0908 D197  ; 报警信号延时, 上料左夹爪升降气缸缩回报警
; rung 9
LD 8.14  ; 上料左夹爪升降气缸
ANDNOT T0008  ; 上料左夹爪升降气缸伸出位延时
TIMX(550) 0909 D197  ; 报警信号延时, 上料左夹爪升降气缸伸出报警
; rung 10
LDNOT 8.15  ; 上料右夹爪升降气缸
ANDNOT T0009  ; 上料右升降气缸缩回位
TIMX(550) 0910 D197  ; 报警信号延时, 上料右夹爪升降气缸缩回报警
; rung 11
LD 8.15  ; 上料右夹爪升降气缸
ANDNOT T0010  ; 上料右夹爪升降气缸伸出位延时
TIMX(550) 0911 D197  ; 报警信号延时, 上料右夹爪升降气缸伸出报警
; rung 12
LD 9.00  ; $?St$Bk?_#[1174] / 上料左夹爪气缸 / $?St$Bk?_#[1174]
ANDNOT T0011  ; 上料夹爪1张开位延时
TIMX(550) 0912 D197  ; 报警信号延时, 上料左夹爪张开位报警
; rung 13
LDNOT 9.00  ; $?St$Bk?_#[1174] / 上料左夹爪气缸 / $?St$Bk?_#[1174]
ANDNOT T0012  ; 上料左夹爪夹紧位延时
ANDNOT H0.05  ; 空跑程序-HMI
TIMX(550) 0913 D197  ; 报警信号延时, 上料左夹爪夹紧报警
; rung 14
LD 9.01  ; 上料右夹爪
ANDNOT T0013  ; 上料右夹爪张开位延时
TIMX(550) 0914 D197  ; 报警信号延时, 上料夹爪2张开报警
; rung 15
LDNOT 9.01  ; 上料右夹爪
ANDNOT T0014  ; 上料右夹爪夹紧位延时
ANDNOT H0.05  ; 空跑程序-HMI
TIMX(550) 0915 D197  ; 报警信号延时, 上料夹爪2夹紧报警

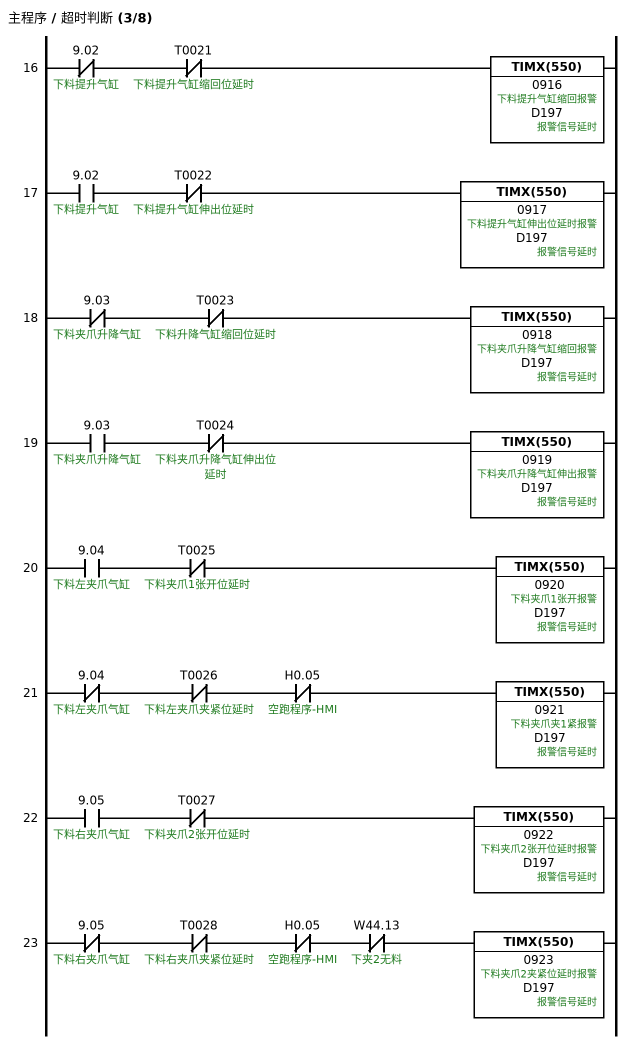
; rung 16
LDNOT 9.02  ; 下料提升气缸
ANDNOT T0021  ; 下料提升气缸缩回位延时
TIMX(550) 0916 D197  ; 报警信号延时, 下料提升气缸缩回报警
; rung 17
LD 9.02  ; 下料提升气缸
ANDNOT T0022  ; 下料提升气缸伸出位延时
TIMX(550) 0917 D197  ; 报警信号延时, 下料提升气缸伸出位延时报警
; rung 18
LDNOT 9.03  ; 下料夹爪升降气缸
ANDNOT T0023  ; 下料升降气缸缩回位延时
TIMX(550) 0918 D197  ; 报警信号延时, 下料夹爪升降气缸缩回报警
; rung 19
LD 9.03  ; 下料夹爪升降气缸
ANDNOT T0024  ; 下料夹爪升降气缸伸出位延时
TIMX(550) 0919 D197  ; 报警信号延时, 下料夹爪升降气缸伸出报警
; rung 20
LD 9.04  ; 下料左夹爪气缸
ANDNOT T0025  ; 下料夹爪1张开位延时
TIMX(550) 0920 D197  ; 报警信号延时, 下料夹爪1张开报警
; rung 21
LDNOT 9.04  ; 下料左夹爪气缸
ANDNOT T0026  ; 下料左夹爪夹紧位延时
ANDNOT H0.05  ; 空跑程序-HMI
TIMX(550) 0921 D197  ; 报警信号延时, 下料夹爪夹1紧报警
; rung 22
LD 9.05  ; 下料右夹爪气缸
ANDNOT T0027  ; 下料夹爪2张开位延时
TIMX(550) 0922 D197  ; 报警信号延时, 下料夹爪2张开位延时报警
; rung 23
LDNOT 9.05  ; 下料右夹爪气缸
ANDNOT T0028  ; 下料右夹爪夹紧位延时
ANDNOT H0.05  ; 空跑程序-HMI
ANDNOT W44.13  ; 下夹2无料
TIMX(550) 0923 D197  ; 报警信号延时, 下料夹爪2夹紧位延时报警

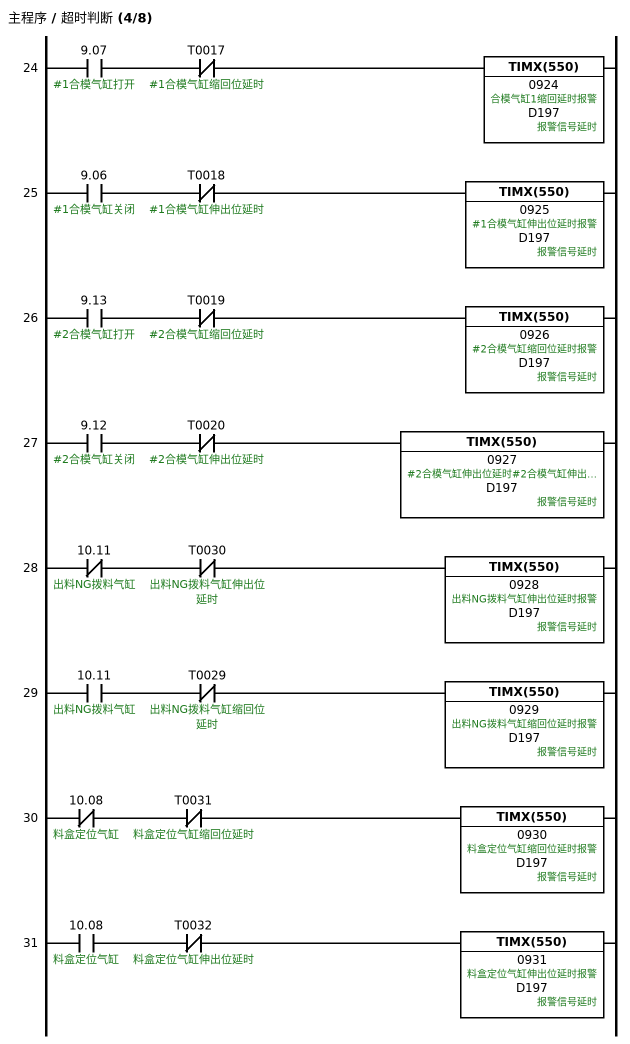
; rung 24
LD 9.07  ; #1合模气缸打开
ANDNOT T0017  ; #1合模气缸缩回位延时
TIMX(550) 0924 D197  ; 报警信号延时, 合模气缸1缩回延时报警
; rung 25
LD 9.06  ; #1合模气缸关闭
ANDNOT T0018  ; #1合模气缸伸出位延时
TIMX(550) 0925 D197  ; 报警信号延时, #1合模气缸伸出位延时报警
; rung 26
LD 9.13  ; #2合模气缸打开
ANDNOT T0019  ; #2合模气缸缩回位延时
TIMX(550) 0926 D197  ; 报警信号延时, #2合模气缸缩回位延时报警
; rung 27
LD 9.12  ; #2合模气缸关闭
ANDNOT T0020  ; #2合模气缸伸出位延时
TIMX(550) 0927 D197  ; 报警信号延时, #2合模气缸伸出位延时#2合模气缸伸出位延时报警
; rung 28
LDNOT 10.11  ; 出料NG拨料气缸
ANDNOT T0030  ; 出料NG拨料气缸伸出位延时
TIMX(550) 0928 D197  ; 报警信号延时, 出料NG拨料气缸伸出位延时报警
; rung 29
LD 10.11  ; 出料NG拨料气缸
ANDNOT T0029  ; 出料NG拨料气缸缩回位延时
TIMX(550) 0929 D197  ; 报警信号延时, 出料NG拨料气缸缩回位延时报警
; rung 30
LDNOT 10.08  ; 料盒定位气缸
ANDNOT T0031  ; 料盒定位气缸缩回位延时
TIMX(550) 0930 D197  ; 报警信号延时, 料盒定位气缸缩回位延时报警
; rung 31
LD 10.08  ; 料盒定位气缸
ANDNOT T0032  ; 料盒定位气缸伸出位延时
TIMX(550) 0931 D197  ; 报警信号延时, 料盒定位气缸伸出位延时报警

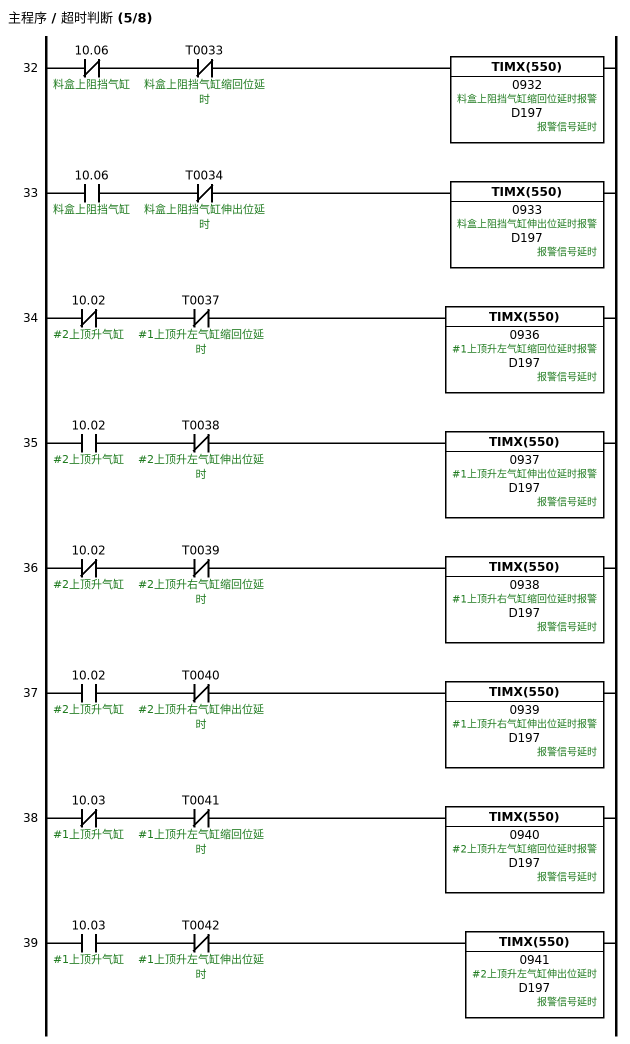
; rung 32
LDNOT 10.06  ; 料盒上阻挡气缸
ANDNOT T0033  ; 料盒上阻挡气缸缩回位延时
TIMX(550) 0932 D197  ; 报警信号延时, 料盒上阻挡气缸缩回位延时报警
; rung 33
LD 10.06  ; 料盒上阻挡气缸
ANDNOT T0034  ; 料盒上阻挡气缸伸出位延时
TIMX(550) 0933 D197  ; 报警信号延时, 料盒上阻挡气缸伸出位延时报警
; rung 34
LDNOT 10.02  ; #2上顶升气缸
ANDNOT T0037  ; #1上顶升左气缸缩回位延时
TIMX(550) 0936 D197  ; 报警信号延时, #1上顶升左气缸缩回位延时报警
; rung 35
LD 10.02  ; #2上顶升气缸
ANDNOT T0038  ; #2上顶升左气缸伸出位延时
TIMX(550) 0937 D197  ; 报警信号延时, #1上顶升左气缸伸出位延时报警
; rung 36
LDNOT 10.02  ; #2上顶升气缸
ANDNOT T0039  ; #2上顶升右气缸缩回位延时
TIMX(550) 0938 D197  ; 报警信号延时, #1上顶升右气缸缩回位延时报警
; rung 37
LD 10.02  ; #2上顶升气缸
ANDNOT T0040  ; #2上顶升右气缸伸出位延时
TIMX(550) 0939 D197  ; 报警信号延时, #1上顶升右气缸伸出位延时报警
; rung 38
LDNOT 10.03  ; #1上顶升气缸
ANDNOT T0041  ; #1上顶升左气缸缩回位延时
TIMX(550) 0940 D197  ; 报警信号延时, #2上顶升左气缸缩回位延时报警
; rung 39
LD 10.03  ; #1上顶升气缸
ANDNOT T0042  ; #1上顶升左气缸伸出位延时
TIMX(550) 0941 D197  ; 报警信号延时, #2上顶升左气缸伸出位延时

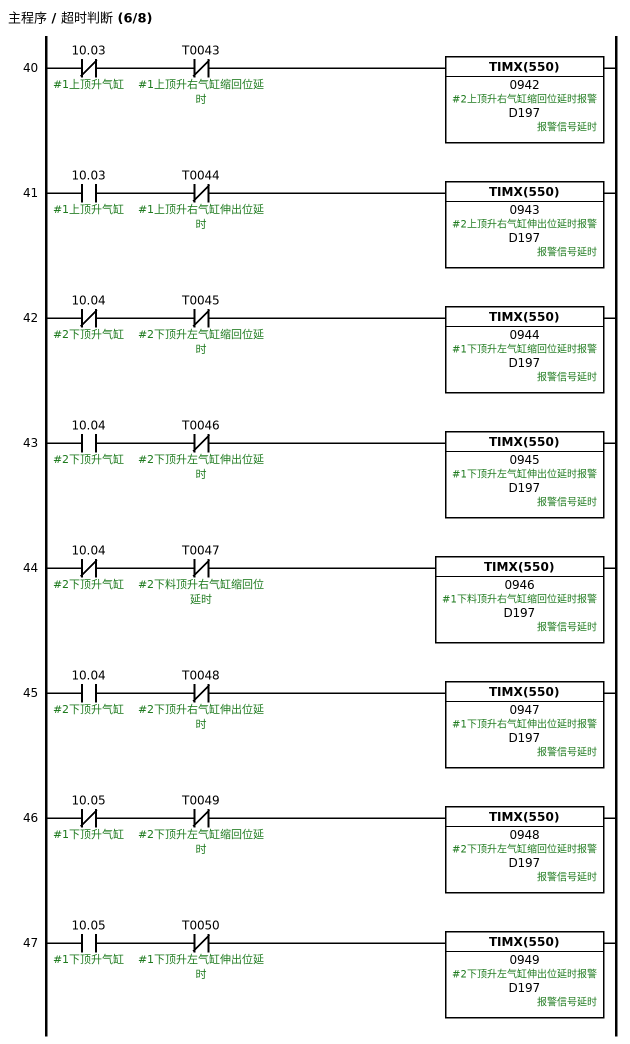
; rung 40
LDNOT 10.03  ; #1上顶升气缸
ANDNOT T0043  ; #1上顶升右气缸缩回位延时
TIMX(550) 0942 D197  ; 报警信号延时, #2上顶升右气缸缩回位延时报警
; rung 41
LD 10.03  ; #1上顶升气缸
ANDNOT T0044  ; #1上顶升右气缸伸出位延时
TIMX(550) 0943 D197  ; 报警信号延时, #2上顶升右气缸伸出位延时报警
; rung 42
LDNOT 10.04  ; #2下顶升气缸
ANDNOT T0045  ; #2下顶升左气缸缩回位延时
TIMX(550) 0944 D197  ; 报警信号延时, #1下顶升左气缸缩回位延时报警
; rung 43
LD 10.04  ; #2下顶升气缸
ANDNOT T0046  ; #2下顶升左气缸伸出位延时
TIMX(550) 0945 D197  ; 报警信号延时, #1下顶升左气缸伸出位延时报警
; rung 44
LDNOT 10.04  ; #2下顶升气缸
ANDNOT T0047  ; #2下料顶升右气缸缩回位延时
TIMX(550) 0946 D197  ; 报警信号延时, #1下料顶升右气缸缩回位延时报警
; rung 45
LD 10.04  ; #2下顶升气缸
ANDNOT T0048  ; #2下顶升右气缸伸出位延时
TIMX(550) 0947 D197  ; 报警信号延时, #1下顶升右气缸伸出位延时报警
; rung 46
LDNOT 10.05  ; #1下顶升气缸
ANDNOT T0049  ; #2下顶升左气缸缩回位延时
TIMX(550) 0948 D197  ; 报警信号延时, #2下顶升左气缸缩回位延时报警
; rung 47
LD 10.05  ; #1下顶升气缸
ANDNOT T0050  ; #1下顶升左气缸伸出位延时
TIMX(550) 0949 D197  ; 报警信号延时, #2下顶升左气缸伸出位延时报警

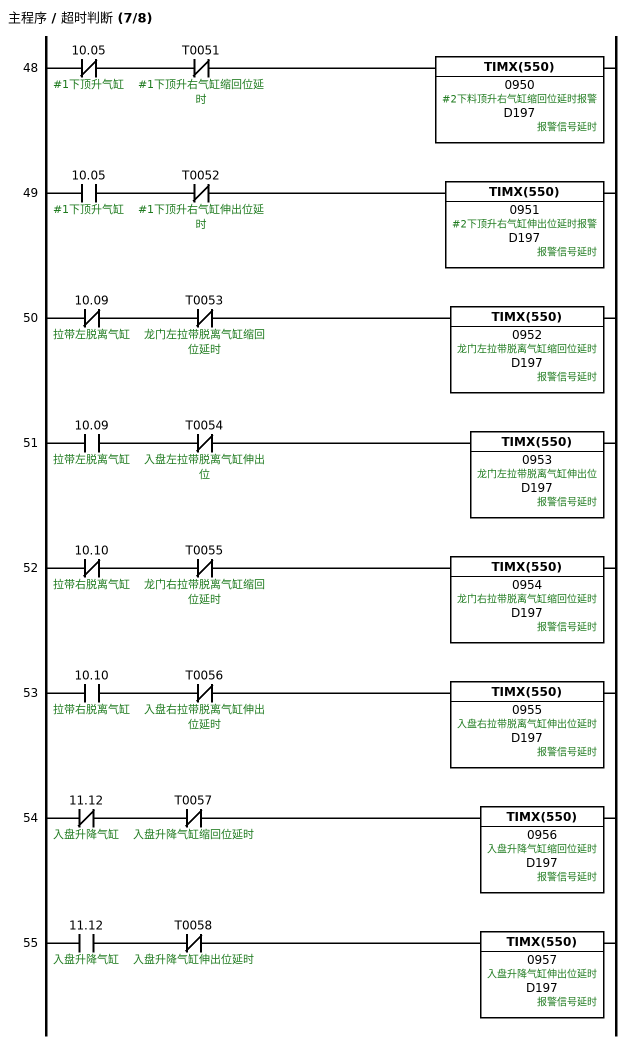
; rung 48
LDNOT 10.05  ; #1下顶升气缸
ANDNOT T0051  ; #1下顶升右气缸缩回位延时
TIMX(550) 0950 D197  ; 报警信号延时, #2下料顶升右气缸缩回位延时报警
; rung 49
LD 10.05  ; #1下顶升气缸
ANDNOT T0052  ; #1下顶升右气缸伸出位延时
TIMX(550) 0951 D197  ; 报警信号延时, #2下顶升右气缸伸出位延时报警
; rung 50
LDNOT 10.09  ; 拉带左脱离气缸
ANDNOT T0053  ; 龙门左拉带脱离气缸缩回位延时
TIMX(550) 0952 D197  ; 报警信号延时, 龙门左拉带脱离气缸缩回位延时
; rung 51
LD 10.09  ; 拉带左脱离气缸
ANDNOT T0054  ; 入盘左拉带脱离气缸伸出位
TIMX(550) 0953 D197  ; 报警信号延时, 龙门左拉带脱离气缸伸出位
; rung 52
LDNOT 10.10  ; 拉带右脱离气缸
ANDNOT T0055  ; 龙门右拉带脱离气缸缩回位延时
TIMX(550) 0954 D197  ; 报警信号延时, 龙门右拉带脱离气缸缩回位延时
; rung 53
LD 10.10  ; 拉带右脱离气缸
ANDNOT T0056  ; 入盘右拉带脱离气缸伸出位延时
TIMX(550) 0955 D197  ; 报警信号延时, 入盘右拉带脱离气缸伸出位延时
; rung 54
LDNOT 11.12  ; 入盘升降气缸
ANDNOT T0057  ; 入盘升降气缸缩回位延时
TIMX(550) 0956 D197  ; 报警信号延时, 入盘升降气缸缩回位延时
; rung 55
LD 11.12  ; 入盘升降气缸
ANDNOT T0058  ; 入盘升降气缸伸出位延时
TIMX(550) 0957 D197  ; 报警信号延时, 入盘升降气缸伸出位延时

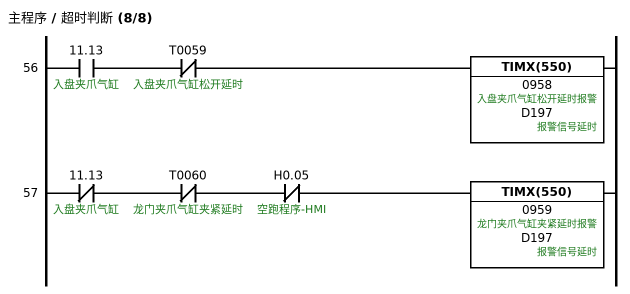
; rung 56
LD 11.13  ; 入盘夹爪气缸
ANDNOT T0059  ; 入盘夹爪气缸松开延时
TIMX(550) 0958 D197  ; 报警信号延时, 入盘夹爪气缸松开延时报警
; rung 57
LDNOT 11.13  ; 入盘夹爪气缸
ANDNOT T0060  ; 龙门夹爪气缸夹紧延时
ANDNOT H0.05  ; 空跑程序-HMI
TIMX(550) 0959 D197  ; 报警信号延时, 龙门夹爪气缸夹紧延时报警

### Section PC交互

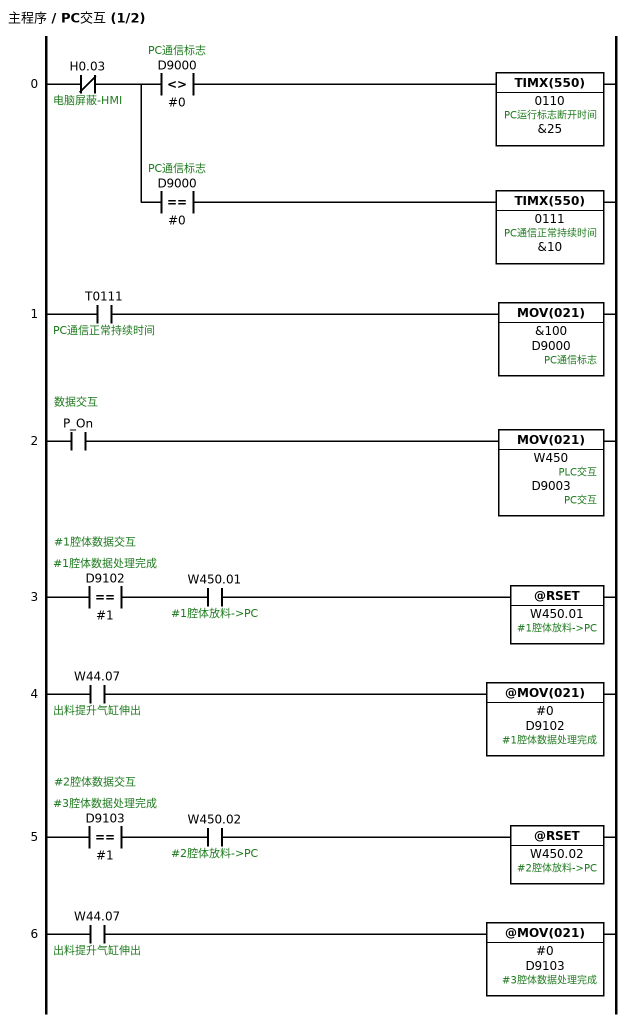
; rung 0
LDNOT H0.03  ; 电脑屏蔽-HMI
OUT TR0
AND<>(305) D9000 #0  ; PC通信标志
TIMX(550) 0110 &25  ; PC运行标志断开时间
LD TR0
AND=(300) D9000 #0  ; PC通信标志
TIMX(550) 0111 &10  ; PC通信正常持续时间
; rung 1
LD T0111  ; PC通信正常持续时间
MOV(021) &100 D9000  ; PC通信标志
; rung 2: 数据交互
LD P_On
MOV(021) W450 D9003  ; PLC交互, PC交互
; rung 3: #1腔体数据交互
LD=(300) D9102 #1  ; #1腔体数据处理完成
AND W450.01  ; #1腔体放料->PC
@RSET W450.01  ; #1腔体放料->PC
; rung 4
LD W44.07  ; 出料提升气缸伸出
@MOV(021) #0 D9102  ; #1腔体数据处理完成
; rung 5: #2腔体数据交互
LD=(300) D9103 #1  ; #3腔体数据处理完成
AND W450.02  ; #2腔体放料->PC
@RSET W450.02  ; #2腔体放料->PC
; rung 6
LD W44.07  ; 出料提升气缸伸出
@MOV(021) #0 D9103  ; #3腔体数据处理完成

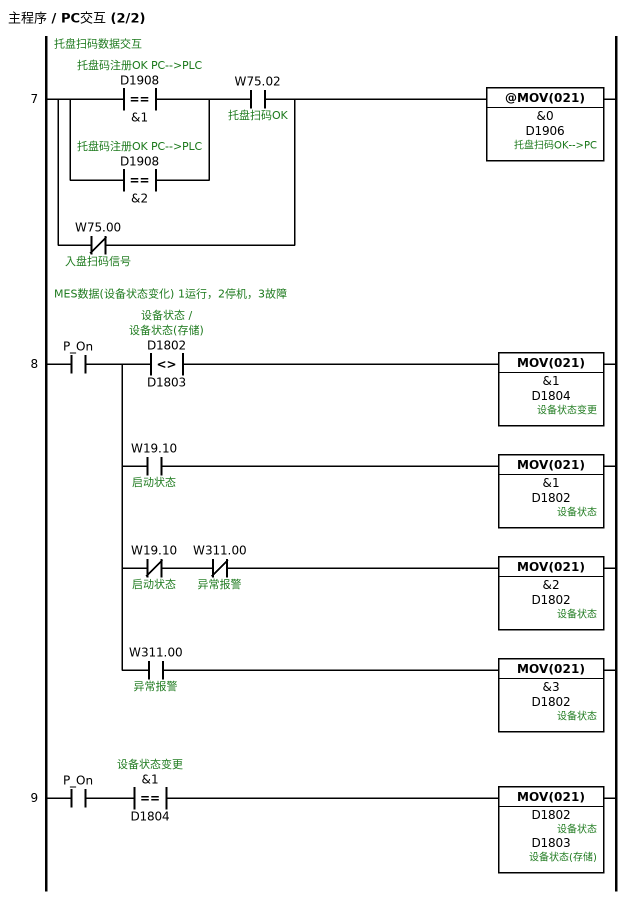
; rung 7: 托盘扫码数据交互
LD=(300) D1908 &1  ; 托盘码注册OK PC-->PLC
OR=(300) D1908 &2  ; 托盘码注册OK PC-->PLC
AND W75.02  ; 托盘扫码OK
ORNOT W75.00  ; 入盘扫码信号
@MOV(021) &0 D1906  ; 托盘扫码OK-->PC
; rung 8: MES数据(设备状态变化) 1运行，2停机，3故障
LD P_On
OUT TR0
AND<>(305) D1802 D1803  ; 设备状态, 设备状态(存储)
MOV(021) &1 D1804  ; 设备状态变更
LD TR0
AND W19.10  ; 启动状态
MOV(021) &1 D1802  ; 设备状态
LD TR0
ANDNOT W19.10  ; 启动状态
ANDNOT W311.00  ; 异常报警
MOV(021) &2 D1802  ; 设备状态
LD TR0
AND W311.00  ; 异常报警
MOV(021) &3 D1802  ; 设备状态
; rung 9
LD P_On
AND=(300) &1 D1804  ; 设备状态变更
MOV(021) D1802 D1803  ; 设备状态, 设备状态(存储)

### Section I_0输出

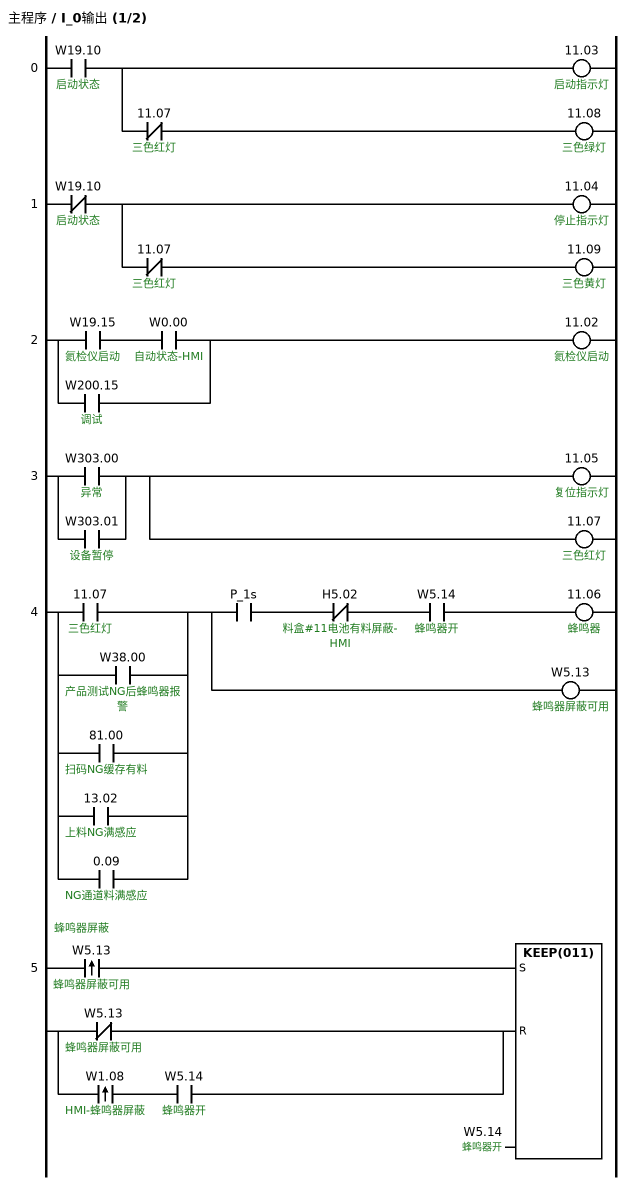
; rung 0
LD W19.10  ; 启动状态
OUT 11.03  ; 启动指示灯
ANDNOT 11.07  ; 三色红灯
OUT 11.08  ; 三色绿灯
; rung 1
LDNOT W19.10  ; 启动状态
OUT 11.04  ; 停止指示灯
ANDNOT 11.07  ; 三色红灯
OUT 11.09  ; 三色黄灯
; rung 2
LD W19.15  ; 氦检仪启动
AND W0.00  ; 自动状态-HMI
OR W200.15  ; 调试
OUT 11.02  ; 氦检仪启动
; rung 3
LD W303.00  ; 异常
OR W303.01  ; 设备暂停
OUT 11.05  ; 复位指示灯
OUT 11.07  ; 三色红灯
; rung 4
LD 11.07  ; 三色红灯
OR W38.00  ; 产品测试NG后蜂鸣器报警
OR 81.00  ; 扫码NG缓存有料
OR 13.02  ; 上料NG满感应
OR 0.09  ; NG通道料满感应
OUT TR0
AND P_1s
ANDNOT H5.02  ; 料盒#11电池有料屏蔽-HMI
AND W5.14  ; 蜂鸣器开
OUT 11.06  ; 蜂鸣器
LD TR0
OUT W5.13  ; 蜂鸣器屏蔽可用
; rung 5: 蜂鸣器屏蔽
@LD W5.13  ; 蜂鸣器屏蔽可用
LDNOT W5.13  ; 蜂鸣器屏蔽可用
@LD W1.08  ; HMI-蜂鸣器屏蔽
AND W5.14  ; 蜂鸣器开
ORLD
KEEP(011) W5.14  ; 蜂鸣器开

